FUNCTION_BLOCK AR_DEADBAND_COMPARE (* Vergleicht einen REAL-Messwert gegen ein Fenster [WINDOW_MIN, WINDOW_MAX]: ABOVE (Y > WINDOW_MAX), BELOW (Y < WINDOW_MIN), CENTERED (dazwischen). Fuer ein symmetrisches Totband um Null WINDOW_MIN=-Totband/WINDOW_MAX=+Totband setzen (z.B. Lenkwinkel-Zentrierung); genauso fuer ein beliebiges Fenster nutzbar (z.B. Farbgrenzen). Jedes Plug feuert sein Event bei Y-Aenderung nur, wenn sich sein eigener Wert tatsaechlich aendert (nicht bei jedem Y-Update alle drei); bei WINDOW_MIN/WINDOW_MAX-Aenderung (in der Praxis meist nur einmal beim Start) werden der Einfachheit halber immer alle drei neu gesetzt. *)
  (* Standard: 61499-2; Description: Fenstervergleich / Totbandauswertung für AR-Messwerte (ABOVE, BELOW, CENTERED) *)
  (* Version 2.0, 2026-09-11, Franz Höpfinger, Verallgemeinert von symmetrischem Totband (1 DEADBAND-Socket) auf beliebiges Fenster (WINDOW_MIN/WINDOW_MAX) - z.B. fuer FillWindowFS_AR nutzbar. Y-Aenderung setzt ABOVE/BELOW/CENTERED jetzt nur noch einzeln bei tatsaechlicher Aenderung (vorher immer alle drei). *)
  (* Version 1.1, 2026-09-11, Franz Höpfinger, DEADBAND von InputVar auf AR-Socket umgestellt (konsistent mit Y) - fester Wert weiterhin ueber adapter::types::unidirectional::AR::initval::initval_AR moeglich *)
  (* Version 1.0, 2026-09-11, Franz Höpfinger, initial implementation - fuer Achslenkung-Mittelpunkt-Automatik, generisch fuer jede Totband-Zentrierung (z.B. spaeter Hangausgleich) *)
  PACKAGE adapter::Engineering::measurements;
  (* Documentation:
  Fenstervergleich / Totbandauswertung (AR_DEADBAND_COMPARE)
   Der Funktionsbaustein AR_DEADBAND_COMPARE vergleicht einen analogen Messwert Y (über ein AR-Adapter-Socket) dynamisch gegen ein definiertes Wertefenster [WINDOW_MIN, WINDOW_MAX].
   Ausgangs-Plugs (AX)
    - ABOVE: Geht auf TRUE, wenn Y > WINDOW_MAX.
   - CENTERED: Geht auf TRUE, wenn WINDOW_MIN <= Y <= WINDOW_MAX (Messwert im Totband / Fenster).
   - BELOW: Geht auf TRUE, wenn Y < WINDOW_MIN.
    Eingangs-Sockets (AR)
    - Y: Analoger Eingangsmesswert.
   - WINDOW_MIN: Untere Fenstergrenze (z. B. negatives Totband -DEADBAND oder unterer Schwellwert).
   - WINDOW_MAX: Obere Fenstergrenze (z. B. positives Totband +DEADBAND oder oberer Schwellwert).
    Ereignis-Verhalten
   Bei einer Änderung des Messwerts Y lösen nur diejenigen Plugs ein Ereignis aus, deren boolescher Zustand sich tatsächlich geändert hat (ereignisdiskrete Effizienz). Bei einer Änderung von WINDOW_MIN oder WINDOW_MAX werden alle drei Ausgänge neu berechnet und aktualisiert.
   Anwendungsszenarien
    - Lenkwinkel-Mittelpunktzentrierung: Überprüfung, ob sich ein Lenksensor innerhalb des Totbandes um 0° befindet (WINDOW_MIN = -Totband, WINDOW_MAX = +Totband).
   - Fenster- / Hysterese-Überwachung: Auswertung von Grenzwert- oder Farbbereichen (z. B. grün/rot in Visualisierungen).
  *)
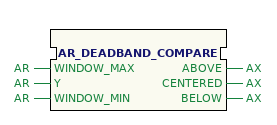
  SOCKETS
    WINDOW_MAX : adapter::types::unidirectional::AR; (* AR-Socket (Eingang): Obere Fenstergrenze (z. B. +Totband oder oberer Grenzwert) *)
    Y : adapter::types::unidirectional::AR; (* AR-Socket (Eingang): Zu vergleichender Eingangsmesswert *)
    WINDOW_MIN : adapter::types::unidirectional::AR; (* AR-Socket (Eingang): Untere Fenstergrenze (z. B. -Totband oder unterer Grenzwert) *)
  END_SOCKETS
  PLUGS
    ABOVE : adapter::types::unidirectional::AX; (* AX-Plug (Ausgang): TRUE wenn Messwert Y > WINDOW_MAX, Ereignis E1 nur bei Zustandsänderung *)
    CENTERED : adapter::types::unidirectional::AX; (* AX-Plug (Ausgang): TRUE wenn WINDOW_MIN <= Y <= WINDOW_MAX (im Fenster/Totband), Ereignis E1 nur bei Zustandsänderung *)
    BELOW : adapter::types::unidirectional::AX; (* AX-Plug (Ausgang): TRUE wenn Messwert Y < WINDOW_MIN, Ereignis E1 nur bei Zustandsänderung *)
  END_PLUGS
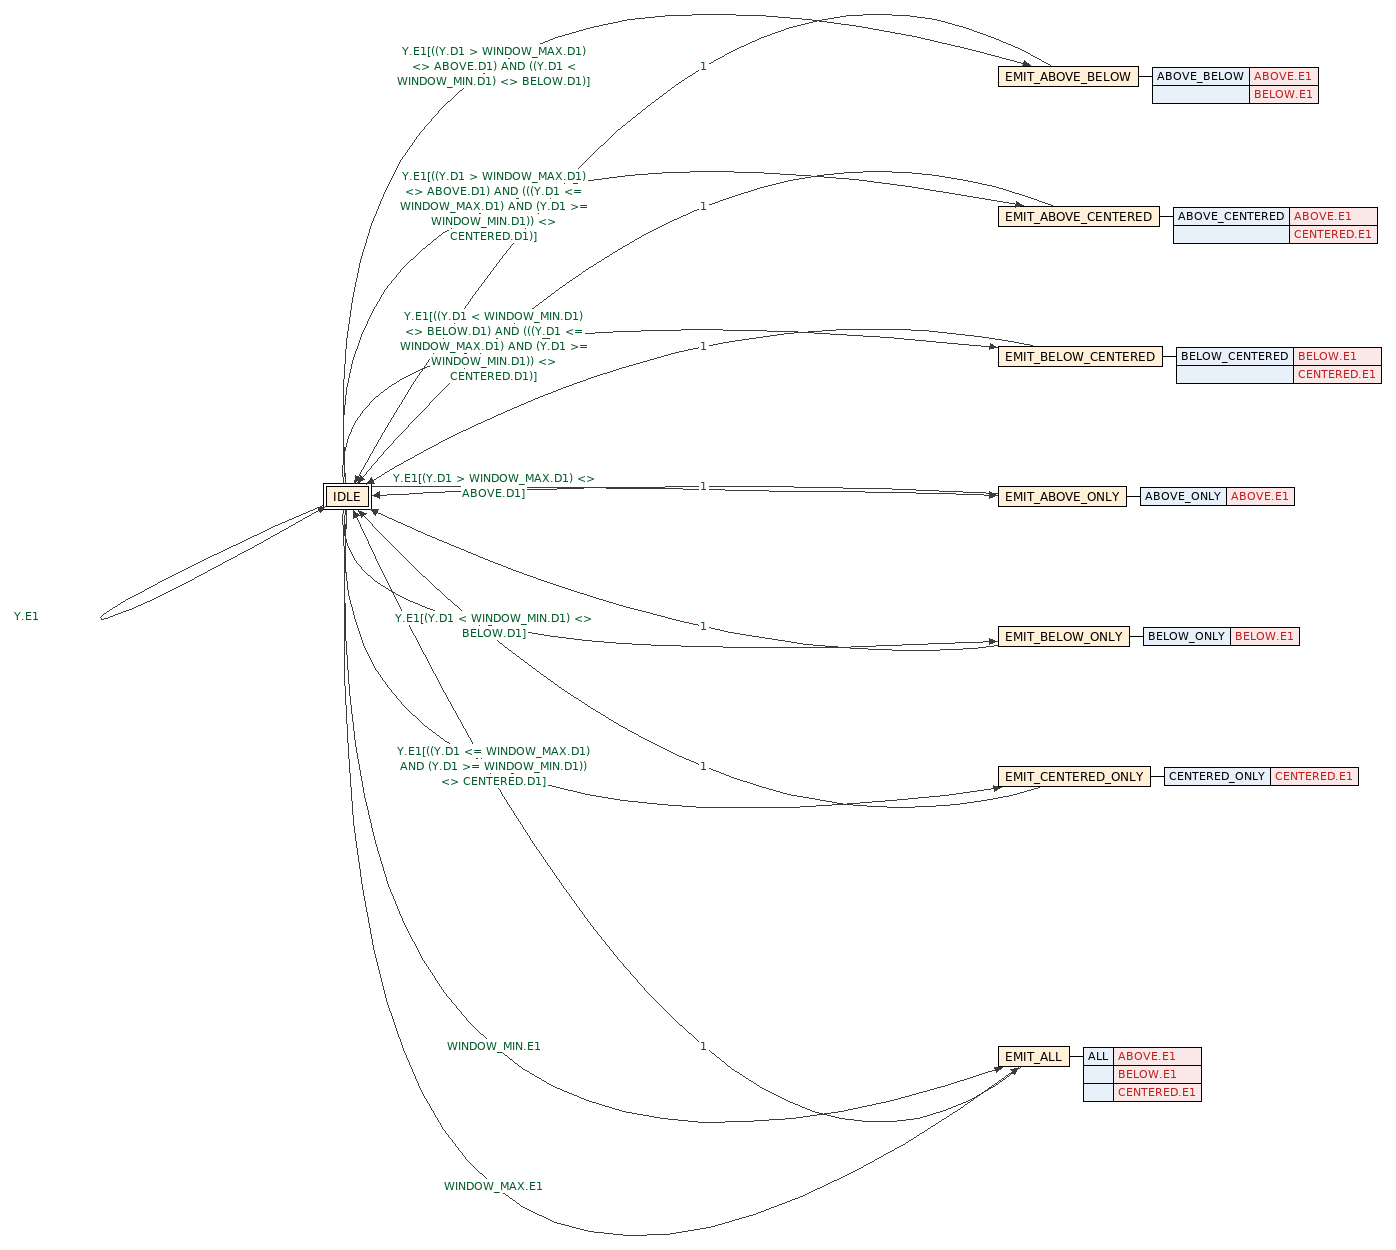
  EC_STATES
    IDLE; (* Ruhezustand – Wartet auf Ereignisse an Y.E1, WINDOW_MIN.E1 oder WINDOW_MAX.E1 *)
    EMIT_ABOVE_BELOW : ABOVE_BELOW -> ABOVE.E1, -> BELOW.E1; (* Aktualisiert ABOVE und BELOW und sendet E1-Ereignisse an beide Plugs *)
    EMIT_ABOVE_CENTERED : ABOVE_CENTERED -> ABOVE.E1, -> CENTERED.E1; (* Aktualisiert ABOVE und CENTERED und sendet E1-Ereignisse an beide Plugs *)
    EMIT_BELOW_CENTERED : BELOW_CENTERED -> BELOW.E1, -> CENTERED.E1; (* Aktualisiert BELOW und CENTERED und sendet E1-Ereignisse an beide Plugs *)
    EMIT_ABOVE_ONLY : ABOVE_ONLY -> ABOVE.E1; (* Aktualisiert nur ABOVE und sendet E1-Ereignis an ABOVE *)
    EMIT_BELOW_ONLY : BELOW_ONLY -> BELOW.E1; (* Aktualisiert nur BELOW und sendet E1-Ereignis an BELOW *)
    EMIT_CENTERED_ONLY : CENTERED_ONLY -> CENTERED.E1; (* Aktualisiert nur CENTERED und sendet E1-Ereignis an CENTERED *)
    EMIT_ALL : ALL -> ABOVE.E1, -> BELOW.E1, -> CENTERED.E1; (* Aktualisiert ABOVE, BELOW sowie CENTERED und sendet E1-Ereignisse an alle drei Plugs (z. B. bei Fenstergrenzenänderung) *)
  END_STATES
  EC_TRANSITIONS
    IDLE TO EMIT_ABOVE_BELOW := Y.E1[((Y.D1 > WINDOW_MAX.D1) <> ABOVE.D1) AND ((Y.D1 < WINDOW_MIN.D1) <> BELOW.D1)];
    IDLE TO EMIT_ABOVE_CENTERED := Y.E1[((Y.D1 > WINDOW_MAX.D1) <> ABOVE.D1) AND (((Y.D1 <= WINDOW_MAX.D1) AND (Y.D1 >= WINDOW_MIN.D1)) <> CENTERED.D1)];
    IDLE TO EMIT_BELOW_CENTERED := Y.E1[((Y.D1 < WINDOW_MIN.D1) <> BELOW.D1) AND (((Y.D1 <= WINDOW_MAX.D1) AND (Y.D1 >= WINDOW_MIN.D1)) <> CENTERED.D1)];
    IDLE TO EMIT_ABOVE_ONLY := Y.E1[(Y.D1 > WINDOW_MAX.D1) <> ABOVE.D1];
    IDLE TO EMIT_BELOW_ONLY := Y.E1[(Y.D1 < WINDOW_MIN.D1) <> BELOW.D1];
    IDLE TO EMIT_CENTERED_ONLY := Y.E1[((Y.D1 <= WINDOW_MAX.D1) AND (Y.D1 >= WINDOW_MIN.D1)) <> CENTERED.D1];
    IDLE TO IDLE := Y.E1;
    IDLE TO EMIT_ALL := WINDOW_MIN.E1;
    IDLE TO EMIT_ALL := WINDOW_MAX.E1;
    EMIT_ABOVE_BELOW TO IDLE := 1;
    EMIT_ABOVE_CENTERED TO IDLE := 1;
    EMIT_BELOW_CENTERED TO IDLE := 1;
    EMIT_ABOVE_ONLY TO IDLE := 1;
    EMIT_BELOW_ONLY TO IDLE := 1;
    EMIT_CENTERED_ONLY TO IDLE := 1;
    EMIT_ALL TO IDLE := 1;
  END_TRANSITIONS
  ALGORITHM ABOVE_BELOW IN ST: (* Berechnet ABOVE (Y > WINDOW_MAX) und BELOW (Y < WINDOW_MIN) *)
ABOVE.D1 := Y.D1 > WINDOW_MAX.D1;
BELOW.D1 := Y.D1 < WINDOW_MIN.D1;
  END_ALGORITHM
  ALGORITHM ABOVE_CENTERED IN ST: (* Berechnet ABOVE (Y > WINDOW_MAX) und CENTERED (WINDOW_MIN <= Y <= WINDOW_MAX) *)
ABOVE.D1 := Y.D1 > WINDOW_MAX.D1;
CENTERED.D1 := (Y.D1 <= WINDOW_MAX.D1) AND (Y.D1 >= WINDOW_MIN.D1);
  END_ALGORITHM
  ALGORITHM BELOW_CENTERED IN ST: (* Berechnet BELOW (Y < WINDOW_MIN) und CENTERED (WINDOW_MIN <= Y <= WINDOW_MAX) *)
BELOW.D1 := Y.D1 < WINDOW_MIN.D1;
CENTERED.D1 := (Y.D1 <= WINDOW_MAX.D1) AND (Y.D1 >= WINDOW_MIN.D1);
  END_ALGORITHM
  ALGORITHM ABOVE_ONLY IN ST: (* Berechnet ABOVE (Y > WINDOW_MAX) *)
ABOVE.D1 := Y.D1 > WINDOW_MAX.D1;
  END_ALGORITHM
  ALGORITHM BELOW_ONLY IN ST: (* Berechnet BELOW (Y < WINDOW_MIN) *)
BELOW.D1 := Y.D1 < WINDOW_MIN.D1;
  END_ALGORITHM
  ALGORITHM CENTERED_ONLY IN ST: (* Berechnet CENTERED (WINDOW_MIN <= Y <= WINDOW_MAX) *)
CENTERED.D1 := (Y.D1 <= WINDOW_MAX.D1) AND (Y.D1 >= WINDOW_MIN.D1);
  END_ALGORITHM
  ALGORITHM ALL IN ST: (* Berechnet alle Ausgänge: ABOVE, BELOW und CENTERED *)
ABOVE.D1 := Y.D1 > WINDOW_MAX.D1;
BELOW.D1 := Y.D1 < WINDOW_MIN.D1;
CENTERED.D1 := (Y.D1 <= WINDOW_MAX.D1) AND (Y.D1 >= WINDOW_MIN.D1);
  END_ALGORITHM
END_FUNCTION_BLOCK
